(* CoDeSys 2.3 export: INVALARM_FB.EXP *)

(* POU FB/ФБ аварий/InvAlarm_FB, ST *)
FUNCTION_BLOCK InvAlarm_FB
VAR_INPUT
	inversion: BOOL;
END_VAR
VAR_OUTPUT
	bError: BOOL;
END_VAR
VAR
	TON1 : TON;
	SEMA1 : SEMA;
END_VAR
ton1.IN := SEL (inversion, TRUE, FALSE);  (*инверсия*)

TON1(PT:= T#3s); (*пака  IN=false  на Q=false, как только IN=true через заданое время PT на Q появится true *)

SEMA1(
	CLAIM:=ton1.Q ,
	RELEASE:=b0x0); (*if CLAIM=true of SUSY=true, RELEASE reset. Reset возможен только когда   CLAIM=false*)

bError := SEL (SEMA1.BUSY, FALSE, TRUE);
END_FUNCTION_BLOCK
